# B&R Automation Studio project Lab1
Automation Studio 4.5.2.102

## Logical view

Binary libraries used (declarations not repeated): operator, runtime, astime, AsIecCon, Library

### Package Logical/Libraries - Global libraries

### Library Logical/Libraries/Library (ANSIC)

#### Library.fun - Exported functions and function blocks
```iecst
{REDUND_ERROR} FUNCTION_BLOCK FB_integrator (*TODO: Add your comment here*) (*$GROUP=User,$CAT=User,$GROUPICON=User.png,$CATICON=User.png*)
	VAR_INPUT
		in : REAL;
	END_VAR
	VAR_OUTPUT
		out : REAL;
	END_VAR
	VAR
		dt : REAL;
	END_VAR
END_FUNCTION_BLOCK

{REDUND_ERROR} FUNCTION_BLOCK FB_motor (*TODO: Add your comment here*) (*$GROUP=User,$CAT=User,$GROUPICON=User.png,$CATICON=User.png*)
	VAR_INPUT
		u : REAL;
	END_VAR
	VAR_OUTPUT
		w : REAL;
		phi : REAL;
	END_VAR
	VAR
		integrator : FB_integrator;
		Tm : REAL;
		ke : REAL;
		dt : REAL;
	END_VAR
END_FUNCTION_BLOCK

{REDUND_ERROR} FUNCTION_BLOCK FB_regulator (*TODO: Add your comment here*) (*$GROUP=User,$CAT=User,$GROUPICON=User.png,$CATICON=User.png*)
	VAR_INPUT
		e : REAL;
	END_VAR
	VAR_OUTPUT
		u : REAL;
	END_VAR
	VAR
		k_p : REAL;
		k_i : REAL;
		integrator : FB_integrator;
		iyOld : REAL;
		max_abs_value : REAL;
		dt : REAL;
		e_kp : REAL;
	END_VAR
END_FUNCTION_BLOCK
```

#### FB_integrator.c
```c
#include <bur/plctypes.h>
#ifdef __cplusplus
	extern "C"
	{
#endif
	#include "Library.h"
#ifdef __cplusplus
	};
#endif

/* Integrator function */
void FB_integrator(struct FB_integrator* inst)
{
	inst->out += inst->in;
}
```

#### FB_motor.c
```c
#include <bur/plctypes.h>
#ifdef __cplusplus
	extern "C"
	{
#endif
	#include "Library.h"
#ifdef __cplusplus
	};
#endif

/* Motor function */
void FB_motor(struct FB_motor* inst)
{
	inst->integrator.in = (inst->u*(1/inst->ke) - inst->w)*(inst->dt/inst->Tm);
	FB_integrator(&(inst->integrator));
	inst->w = inst->integrator.out;

	inst->integrator.in = inst->w*inst->dt;
	FB_integrator(&(inst->integrator));
	inst->phi = inst->integrator.out;
}
```

#### FB_regulator.c
```c
#include <bur/plctypes.h>
#ifdef __cplusplus
	extern "C"
	{
#endif
	#include "Library.h"
#ifdef __cplusplus
	};
#endif

/* Regulator function */
void FB_regulator(struct FB_regulator* inst)
{
	inst->e_kp = inst->e*inst->k_p;

	inst->integrator.in = inst->e*inst->dt*inst->k_i + inst->iyOld;
	FB_integrator(&(inst->integrator));

	if (inst->e_kp < inst->max_abs_value || inst->e_kp > -inst->max_abs_value);
	else
	{
		if (inst->e_kp > 0)
			inst->e_kp = inst->max_abs_value;
		else
			inst->e_kp = -inst->max_abs_value;
	}

	inst->e_kp += inst->integrator.out;

	if (inst->e_kp < inst->max_abs_value || inst->e_kp > -inst->max_abs_value)
		inst->u = inst->e_kp;
	else
	{
		if (inst->e_kp > 0)
			inst->u = inst->max_abs_value;
		else
			inst->u = -inst->max_abs_value;
	}

	inst->iyOld = inst->u - inst->e_kp;
}
```

### Program Logical/Program (ANSIC)

#### Variables.var
```iecst
VAR
	fb_controller : FB_regulator;
	fb_motor_1 : FB_motor;
	speed : REAL;
	enable : REAL;
	fb_motor_2 : FB_motor;
	count : REAL;
END_VAR
```

#### Cyclic.c
```c
#include <bur/plctypes.h>

#ifdef _DEFAULT_INCLUDES
	#include <AsDefault.h>
#endif

void _CYCLIC ProgramCyclic(void)
{
	if (enable == 1)
	{
		count += 10;
		if (count >= 10000 && count <= 15000)
			speed = 5;
		else
			speed = 0;
	}
	else
		speed = 0;

	fb_controller.e = speed - fb_motor_1.w;
	FB_regulator(&(fb_controller));

	fb_motor_1.u = fb_controller.u;
	fb_motor_2.u = speed;

	FB_motor(&(fb_motor_1));
	FB_motor(&(fb_motor_2));
}
```

#### Init.c
```c
#include <bur/plctypes.h>

#ifdef _DEFAULT_INCLUDES
	#include <AsDefault.h>
#endif

void _INIT ProgramInit(void)
{
	enable = 1;
	count = 0;
	speed = 0;

	fb_controller.dt = 0.002;
	fb_controller.k_i = 160;
	fb_controller.k_p = 6.4;
	fb_controller.max_abs_value = 24;

	fb_motor_1.dt = 0.002;
	fb_motor_1.ke = 160;
	fb_motor_1.Tm = 0.04;

	fb_motor_2.dt = 0.002;
	fb_motor_2.ke = 160;
	fb_motor_2.Tm = 0.04;
}
```

Listed in the project but not available here: Logical/Global.typ, Logical/Global.var, Logical/Libraries/Library/Types.typ, Logical/Libraries/Library/Constants.var
